// SIMATIC S7-200 SMART project (STEP 7-Micro/WIN SMART), CPU ST60

SYMBOL_TABLE 系统符号
First_Scan_On    SM0.1    // 仅在第一个扫描周期时接通
END_SYMBOL_TABLE

ORGANIZATION_BLOCK MAIN:OB1
TITLE=程序注释
BEGIN
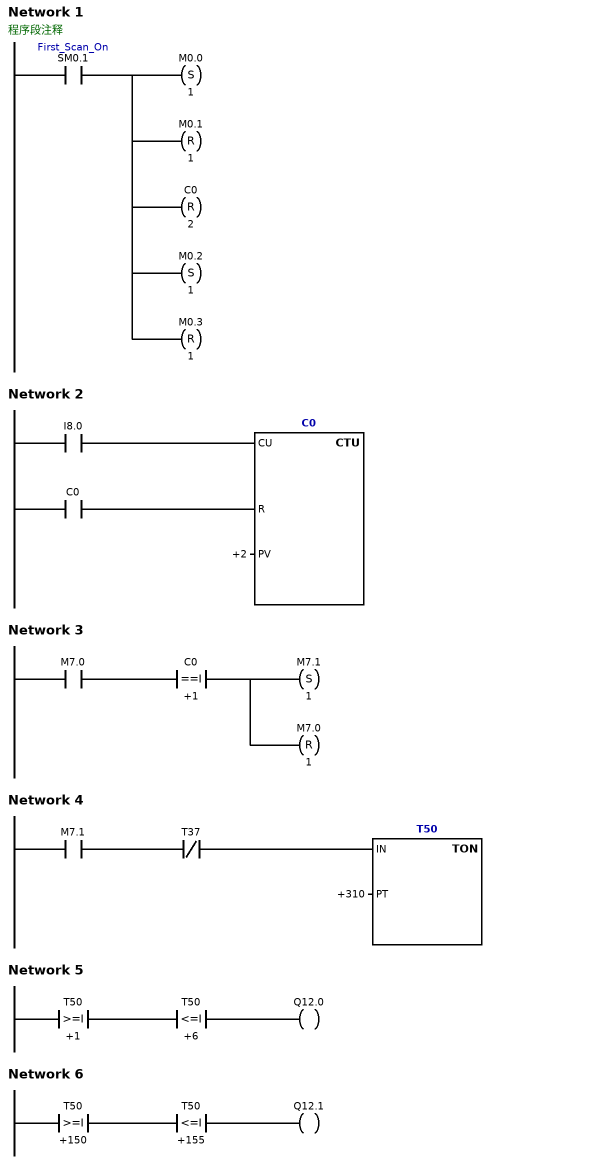
Network 1
// 程序段注释
LD     First_Scan_On:SM0.1
S      M0.0, 1
R      M0.1, 1
R      C0, 2
S      M0.2, 1
R      M0.3, 1
Network 2
LD     I8.0
LD     C0
CTU    C0, +2
Network 3
// (network saved uncompiled; LAD cells follow)
// row 0: c0 -| |- M7.0  c1 -|==I|- C0, +1 v  c2 -(S) M7.1, 1
// row 1: c1 ^  c2 -(R) M7.0, 1
Network 4
// (network saved uncompiled; LAD cells follow)
// row 0: c0 -| |- M7.1  c1 -|/|- T37  c2 --  c3 [TON T50 IN:=power@row0, PT:=+310]
// row 1: c3 [box]
Network 5
// (network saved uncompiled; LAD cells follow)
// row 0: c0 -|>=I|- T50, +1  c1 -|<=I|- T50, +6  c2 -( ) Q12.0
Network 6
// (network saved uncompiled; LAD cells follow)
// row 0: c0 -|>=I|- T50, +150  c1 -|<=I|- T50, +155  c2 -( ) Q12.1
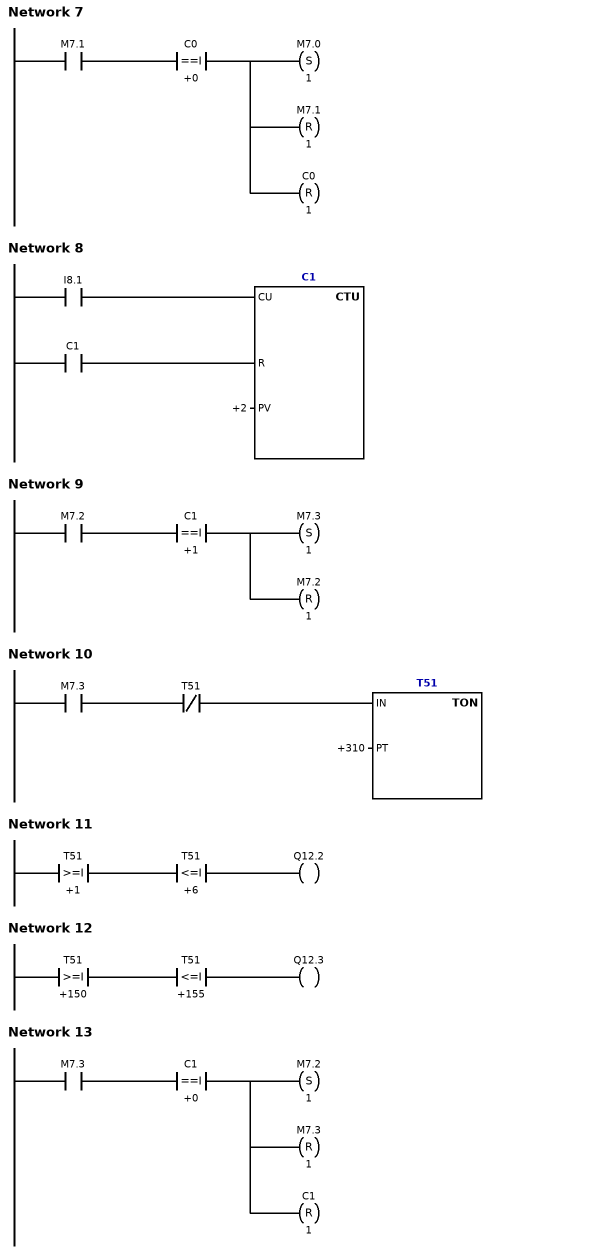
Network 7
// (network saved uncompiled; LAD cells follow)
// row 0: c0 -| |- M7.1  c1 -|==I|- C0, +0 v  c2 -(S) M7.0, 1
// row 1: c1 ^v  c2 -(R) M7.1, 1
// row 2: c1 ^  c2 -(R) C0, 1
Network 8
LD     I8.1
LD     C1
CTU    C1, +2
Network 9
// (network saved uncompiled; LAD cells follow)
// row 0: c0 -| |- M7.2  c1 -|==I|- C1, +1 v  c2 -(S) M7.3, 1
// row 1: c1 ^  c2 -(R) M7.2, 1
Network 10
// (network saved uncompiled; LAD cells follow)
// row 0: c0 -| |- M7.3  c1 -|/|- T51  c2 --  c3 [TON T51 IN:=power@row0, PT:=+310]
// row 1: c3 [box]
Network 11
// (network saved uncompiled; LAD cells follow)
// row 0: c0 -|>=I|- T51, +1  c1 -|<=I|- T51, +6  c2 -( ) Q12.2
Network 12
// (network saved uncompiled; LAD cells follow)
// row 0: c0 -|>=I|- T51, +150  c1 -|<=I|- T51, +155  c2 -( ) Q12.3
Network 13
// (network saved uncompiled; LAD cells follow)
// row 0: c0 -| |- M7.3  c1 -|==I|- C1, +0 v  c2 -(S) M7.2, 1
// row 1: c1 ^v  c2 -(R) M7.3, 1
// row 2: c1 ^  c2 -(R) C1, 1
END_ORGANIZATION_BLOCK
